Staubli VAL3: N15_AproAgafarPuntes.pgx

program N15_AproAgafarPuntes()
  local pointRx l_pAproAgafarPuntes
begin

  // Anar a l'aproximació del punt d'agafar puntes
  if aioGet(aiNumPipeta)==2
    l_pAproAgafarPuntes=pAgafarPuntes8
  else
    l_pAproAgafarPuntes=pAgafarPuntes1
  endIf

  l_pAproAgafarPuntes.trsf.x=l_pAproAgafarPuntes.trsf.x+nXOffset
  l_pAproAgafarPuntes.trsf.y=l_pAproAgafarPuntes.trsf.y+nYOffset
  l_pAproAgafarPuntes.trsf.z=l_pAproAgafarPuntes.trsf.z+nZOffset

  if nZApro>0
    l_pAproAgafarPuntes.trsf.z=l_pAproAgafarPuntes.trsf.z+nZApro
  else
    l_pAproAgafarPuntes.trsf.z=l_pAproAgafarPuntes.trsf.z+100
  endIf

  movel(l_pAproAgafarPuntes,tToolActiva,mLent)
  waitEndMove()

  bTaskDone=true
end
